{attribute 'qualified_only'}
{attribute 'strict'}
TYPE ST_SF3_1_ESTOP :
STRUCT
    bSI_ES_EXP : BOOL;
    bSI_ES_OPT : BOOL;
    bSI_ES_EXT : BOOL;
END_STRUCT
END_TYPE

(* stored: Version 1.1.0.1
   DUT ST_SF3_1_ESTOP: Id {cee9a2af-de4d-0f20-1f26-6c0fafd62275} *)
